FUNCTION_BLOCK FB_MotionAxisNC EXTENDS FB_MotionAxisCommon
VAR_INPUT
END_VAR
VAR_OUTPUT
END_VAR
VAR
    // cathc this from interlock block or send it to interlock block in fb_init or call_after_init
    // catch limit status from motioninterlock block cyclic or just after execHome has pos edge.
    fbHomeMcSetPos: MC_SetPosition;
    fbHomeMcJog: MC_Jog;
    rtHomeExec: R_TRIG;
    ftHomeExec: F_TRIG;
    nHomeStateMachine: E_HomeStates;
    nHomeStateAfterStop: E_HomeStates;
    nHomeMoves: INT;
    bHomeFirstDir: BOOL;
    bAtHome: BOOL;
    bHomeMove: BOOL;
    nHomeErrCount: INT;
END_VAR
VAR CONSTANT
    (*
        This is a simpler way of disabling the soft limits that ends up being really obvious if something has gone wrong.
        If you turn the limits off/on, not only do you need to keep track of if you had soft limits set,
        but you need to always restore this properly or risk some issue.
        Instead, I set position to a ridiculous value that can always move forward or backward.
        If this gets stuck for any reason it's very clear that something has gone wrong,
        rather than a silent failure of the soft limit marks.
    *)
    FWD_START: LREAL := -99999999;
    BWD_START: LREAL :=  99999999;
END_VAR

SUPER^.PreCommon();

THIS^.Home(THIS^.bCommandedMoveHome);

SUPER^.PostCommon();

METHOD Home
VAR_INPUT
    bExecute: BOOL;
END_VAR
THIS^.fbHomeMcSetPos.Options.ClearPositionLag := TRUE;
THIS^.rtHomeExec(CLK:=THIS^.bCommandedMoveHome);
THIS^.ftHomeExec(CLK:=THIS^.bCommandedMoveHome);
THIS^.rtHomeAborted(CLK:=THIS^.bInterrupted);

SUPER^.bHomeError R= NOT THIS^.bCommandedMoveHome;
IF NOT SUPER^.bHomeError THEN
    SUPER^.nHomeErrorID := 0;
END_IF

CASE THIS^.nHomeMode OF
    E_EpicsHomeCmd.LOW_LIMIT:
        THIS^.bHomeFirstDir := FALSE;
        THIS^.bAtHome := NOT THIS^.bLimitBackwardEnable;
        THIS^.bHomeMove := THIS^.bCommandedMoveHome;
    E_EpicsHomeCmd.HIGH_LIMIT:
        THIS^.bHomeFirstDir := TRUE;
        THIS^.bAtHome := NOT THIS^.bLimitForwardEnable;
        THIS^.bHomeMove := THIS^.bCommandedMoveHome;
    E_EpicsHomeCmd.HOME_VIA_LOW:
        THIS^.bHomeFirstDir := FALSE;
        THIS^.bAtHome := bHome;
        THIS^.bHomeMove := THIS^.bCommandedMoveHome;
    E_EpicsHomeCmd.HOME_VIA_HIGH:
        THIS^.bHomeFirstDir := TRUE;
        THIS^.bAtHome := THIS^.bHome;
        THIS^.bHomeMove := THIS^.bCommandedMoveHome;
    E_EpicsHomeCmd.ABSOLUTE_SET:
        THIS^.fbHomeMcSetPos(
            Axis:=AxisRef,
            Execute:=THIS^.bCommandedMoveHome,
            // to review, this should come from EPICS Itf
            Position:=SUPER^.fHomePosition);
        SUPER^.bHomeBusy := THIS^.rtHomeExec.Q;
        SUPER^.bHomeDone := NOT THIS^.rtHomeExec.Q;
        THIS^.bHomeMove := FALSE;
    E_EpicsHomeCmd.NONE:
        THIS^.bHomeMove := FALSE;
        SUPER^.bHomeBusy := THIS^.rtHomeExec.Q;
        SUPER^.bHomeDone := NOT THIS^.rtHomeExec.Q;
    ELSE
        THIS^.bHomeMove := FALSE;
END_CASE

IF THIS^.bHomeMove THEN
    IF THIS^.bHomeBusy AND THIS^.rtHomeAborted.Q THEN
        THIS^.nHomeStateMachine := E_HomeStates.ERROR;
        SUPER^.bHomeInterrupted := TRUE;
    END_IF
    CASE THIS^.nHomeStateMachine OF
        // Wait for a rising edge
        E_HomeStates.IDLE:
            SUPER^.bHomeBusy := FALSE;
            THIS^.nHomeErrCount := 0;
            THIS^.fbHomeMcSetPos(
                Axis:=AxisRef,
                Execute:=FALSE);
            THIS^.fbHomeMcJog(
                Axis:=AxisRef,
                JogForward:=FALSE,
                JogBackwards:=FALSE);
            IF THIS^.rtHomeExec.Q THEN
                THIS^.nHomeStateMachine := E_HomeStates.NEXT_MOVE;
                nHomeMoves := 0;
                SUPER^.bHomeDone := FALSE;
                SUPER^.bHomeBusy := TRUE;
                SUPER^.bHomeError := FALSE;
                SUPER^.nHomeErrorID := 0;
                SUPER^.bHomeInterrupted := FALSE;
            END_IF
        // Figure out whether to move forward, move backward, or give up
        E_HomeStates.NEXT_MOVE:
            THIS^.fbHomeMcSetPos(
                Axis:=AxisRef,
                Execute:=FALSE);
            THIS^.fbHomeMcJog(
                Axis:=AxisRef,
                JogForward:=FALSE,
                JogBackwards:=FALSE);
            CASE nHomeMoves OF
                0:
                    IF THIS^.bHomeFirstDir THEN
                        nHomeStateAfterStop := E_HomeStates.CHECK_FWD;
                    ELSE
                        nHomeStateAfterStop := E_HomeStates.CHECK_BWD;
                    END_IF
                1:
                    IF NOT THIS^.bHomeFirstDir THEN
                        nHomeStateAfterStop := E_HomeStates.CHECK_FWD;
                    ELSE
                        nHomeStateAfterStop := E_HomeStates.CHECK_BWD;
                    END_IF
                ELSE
                    nHomeStateAfterStop := E_HomeStates.ERROR;
            END_CASE
            nHomeMoves := nHomeMoves + 1;
            IF THIS^.bAtHome THEN
                nHomeStateAfterStop := E_HomeStates.FINAL_MOVE;
            END_IF
            THIS^.nHomeStateMachine := E_HomeStates.WAIT_STOP;
        // Move forward until we find the home signal or reach end of travel
        E_HomeStates.CHECK_FWD:
            THIS^.fbHomeMcSetPos(
                Axis:=AxisRef,
                Execute:=TRUE,
                Position:=FWD_START);
            THIS^.fbHomeMcJog(
                Axis:=AxisRef,
                JogForward:=bLimitForwardEnable AND NOT bATHome,
                JogBackwards:=FALSE,
                Mode:=E_JogMode.MC_JOGMODE_CONTINOUS,
                Velocity:=SUPER^.stAxisParameters.fRefVeloSearch);
            IF NOT THIS^.fbHomeMcJog.JogForward THEN
                THIS^.nHomeStateMachine := E_HomeStates.NEXT_MOVE;
            ELSIF THIS^.fbHomeMcJog.Error THEN
                THIS^.fbHomeMcJog(
                    Axis:=AxisRef,
                    JogForward:=FALSE,
                    JogBackwards:=FALSE);
                THIS^.nHomeErrCount := THIS^.nHomeErrCount + 1;
                IF THIS^.nHomeErrCount >= 3 THEN
                    THIS^.nHomeStateMachine := E_HomeStates.ERROR;
                END_IF
            END_IF
        // Move backward until we find the home signal or reach end of travel
        E_HomeStates.CHECK_BWD:
            THIS^.fbHomeMcSetPos(
                Axis:=AxisRef,
                Execute:=TRUE,
                Position:=BWD_START);
            THIS^.fbHomeMcJog(
                Axis:=AxisRef,
                JogForward:=FALSE,
                JogBackwards:=bLimitBackwardEnable AND NOT bAtHome,
                Mode:=E_JogMode.MC_JOGMODE_CONTINOUS,
                Velocity:=SUPER^.stAxisParameters.fRefVeloSearch);
            IF NOT THIS^.fbHomeMcJog.JogBackwards THEN
                THIS^.nHomeStateMachine := E_HomeStates.NEXT_MOVE;
            ELSIF THIS^.fbHomeMcJog.Error THEN
                THIS^.fbHomeMcJog(
                    Axis:=AxisRef,
                    JogForward:=FALSE,
                    JogBackwards:=FALSE);
                THIS^.nHomeErrCount := THIS^.nHomeErrCount + 1;
                IF THIS^.nHomeErrCount >= 3 THEN
                    THIS^.nHomeStateMachine := E_HomeStates.ERROR;
                END_IF
            END_IF
        // Set position to get within soft lims, move slowly off signal
        E_HomeStates.FINAL_MOVE:
            THIS^.fbHomeMcSetPos(
                Axis:=AxisRef,
                Execute:=TRUE,
                Position:=SUPER^.fHomePosition);
            IF THIS^.bAtHome THEN
                THIS^.fbHomeMcJog(
                    Axis:=AxisRef,
                    JogForward:=NOT bHomeFirstDir,
                    JogBackwards:=bHomeFirstDir,
                    Mode:=E_JogMode.MC_JOGMODE_CONTINOUS,
                    Velocity:=SUPER^.stAxisParameters.fRefVeloSync);
            ELSIF THIS^.fbHomeMcJog.Error THEN
                THIS^.fbHomeMcJog(
                    Axis:=AxisRef,
                    JogForward:=FALSE,
                    JogBackwards:=FALSE);
                THIS^.nHomeErrCount := THIS^.nHomeErrCount + 1;
                IF THIS^.nHomeErrCount >= 3 THEN
                    THIS^.nHomeStateMachine := E_HomeStates.ERROR;
                END_IF
            ELSE
                THIS^.fbHomeMcJog(
                    Axis:=AxisRef,
                    JogForward:=FALSE,
                    JogBackwards:=FALSE);
                THIS^.fbHomeMcSetPos(
                    Axis:=AxisRef,
                    Execute:=FALSE);
                THIS^.nHomeStateMachine := E_HomeStates.WAIT_STOP;
                nHomeStateAfterStop := E_HomeStates.FINAL_SETPOS;
            END_IF
        E_HomeStates.FINAL_SETPOS:
            THIS^.fbHomeMcSetPos(
                Axis:=AxisRef,
                Execute:=TRUE,
                Position:=SUPER^.fHomePosition);
            THIS^.nHomeStateMachine := E_HomeStates.IDLE;
            SUPER^.bHomeBusy := FALSE;
            SUPER^.bHomeDone := TRUE;
        E_HomeStates.ERROR:
            SUPER^.bHomeError := TRUE;
            SUPER^.nHomeErrorID := THIS^.fbHomeMcJog.ErrorID;
            nHomeStateMachine := E_HomeStates.FINAL_SETPOS;
            THIS^.fbHomeMcSetPos(
                Axis:=AxisRef,
                Execute:=FALSE);
            IF bHomeInterrupted THEN
                SUPER^.sErrorMessage := 'Homing interrupted';
            ELSE
               SUPER^.sErrorMessage := 'Homing failure';
            END_IF
        E_HomeStates.WAIT_STOP:
            IF AxisRef.Status.NotMoving THEN
                THIS^.nHomeStateMachine := nHomeStateAfterStop;
            END_IF
    END_CASE
END_IF

// we should normally do this in interrupted state if moving
// otherwise we need to reset, the error state should perhaps handle this
IF SUPER^.bCommandedReset THEN
    SUPER^.bHomeBusy := FALSE;
    SUPER^.bHomeDone := FALSE;
    THIS^.bHomeMove := FALSE;
END_IF
END_METHOD

METHOD InterruptMove
END_METHOD

PROPERTY LimBwdEnable : BOOL
GET
LimBwdEnable := bLimitBackwardEnable;
END_GET
SET
bLimitBackwardEnable := LimBwdEnable;
END_SET
END_PROPERTY

PROPERTY LimFwdEnable : BOOL
GET
LimFwdEnable := bLimitForwardEnable;
END_GET
SET
bLimitForwardEnable := LimFwdEnable;
END_SET
END_PROPERTY

PROPERTY LimHome : BOOL
GET
END_GET
SET
END_SET
END_PROPERTY

(*
    Check all post condition before updating bCommandedMoveAbsolute
    The implmentatation will depend on the axis type
    DS402 NC/Direct axis : Implementation need to check that the drive is in the correct mode before initaiting the move then set bCommandedMoveAbsolute
    MP NC axis : will immediately write to bCommandedMoveAbsolute
*)
METHOD StartMove : BOOL
StartMove := SUPER^.StartMove();
END_METHOD

METHOD StopMove
END_METHOD

END_FUNCTION_BLOCK

(* stored: Version 1.1.0.1
   POU FB_MotionAxisNC: Id {c6c45e58-0632-4869-96bd-3ee4e21217a8}, SpecialFunc None
   Method Home: Id {33ae7160-6fd9-4351-881c-ff032354b4f0}
   Method InterruptMove: Id {3b35232d-04d6-4f22-af2c-874d31217d09}
   Property LimBwdEnable: Id {f1c400e3-1909-4392-b56e-42d18fb82eb5}
   Get Get: Id {387cf336-53ef-4887-867f-689596a32728}
   Set Set: Id {3a7e2526-96be-436c-a698-396fafb39ff9}
   Property LimFwdEnable: Id {4be1f54c-a6b2-47bf-8c3c-4d40bc9a1713}
   Get Get: Id {52d07e66-751c-4181-9dfc-b9c3523a2633}
   Set Set: Id {d4c954cf-bea3-4254-a851-6a894af44f6c}
   Property LimHome: Id {2f273079-ccda-4520-984a-f5344492d887}
   Get Get: Id {9dff4bf0-8b8f-4eca-b9a9-23e72d4dbf64}
   Set Set: Id {4a845969-2a16-420f-8c7a-bd49f84481c0}
   Method StartMove: Id {96c9c828-de26-4c5b-86fc-b06f69f3ecce}
   Method StopMove: Id {88a971d1-aaef-4bb6-b7c2-65b47210b532} *)
